FUNCTION_BLOCK FB_Beckhoff_EL5152
VAR_INPUT
	nValue1		: UINT;
	nValue2		: UINT;
END_VAR
VAR
	nControl1		AT %I* : UINT;
	nSetCounter1	AT %I* : UINT;
	nControl2		AT %I* : UINT;
	nSetCounter2	AT %I* : UINT;
	
	nStatus1		AT %Q* : UINT;
	nCounter1		AT %Q* : UINT;	
	nPeriod1    	AT %Q* : UDINT;
	nStatus2		AT %Q* : UINT;
	nCounter2		AT %Q* : UINT;
	nPeriod2    	AT %Q* : UDINT;
END_VAR

nStatus1.2 := nControl1.2;
nStatus2.2 := nControl2.2;

nCounter1 := nValue1;
nCounter2 := nValue2;

PROPERTY INTERNAL Control1 : UINT
SET
nControl1 := Control1;
END_SET
END_PROPERTY

PROPERTY INTERNAL Control2 : UINT
SET
nControl2 := Control2;
END_SET
END_PROPERTY

PROPERTY INTERNAL Counter1 : UINT
GET
Counter1 := nCounter1;
END_GET
END_PROPERTY

PROPERTY INTERNAL Counter2 : UINT
GET
Counter2 := nCounter2;
END_GET
END_PROPERTY

PROPERTY INTERNAL Period1 : UDINT
GET
Period1 := nPeriod1;
END_GET
END_PROPERTY

PROPERTY INTERNAL Period2 : UDINT
GET
Period2 := nPeriod2;
END_GET
END_PROPERTY

PROPERTY INTERNAL SetCounter1 : UINT
SET
nSetCounter1 := SetCounter1;
END_SET
END_PROPERTY

PROPERTY INTERNAL SetCounter2 : UINT
SET
nSetCounter2 := SetCounter2;
END_SET
END_PROPERTY

PROPERTY INTERNAL Status1 : UINT
GET
Status1 := nStatus1;
END_GET
END_PROPERTY

PROPERTY INTERNAL Status2 : UINT
GET
Status2 := nStatus2;
END_GET
END_PROPERTY

END_FUNCTION_BLOCK

(* stored: Version 1.1.0.1, ProductVersion 3.1.4024.12
   POU FB_Beckhoff_EL5152: Id {08baf088-2cf3-00bf-18c7-0387cec0c836}, SpecialFunc None
   Property Control1: Id {5c550402-bb0e-0ef9-0fec-73e14d2bbe4d}
   Set Set: Id {5ba60a83-acbe-0e98-31b5-a65c95cf5871}
   Property Control2: Id {f58e2f72-8d03-0b2d-15ce-8c78cfb46d19}
   Set Set: Id {5db5adfd-c3a6-0ac0-1eea-674a8bd0d24d}
   Property Counter1: Id {03127839-0093-03b2-0a6f-88166eb755f6}
   Get Get: Id {1ff40a2f-399d-0c65-15d8-0c3b4f2bcaeb}
   Property Counter2: Id {1854e639-ce6e-0901-076f-d57c64553137}
   Get Get: Id {3a7e0597-34bc-0eb5-0cc1-6255b4e03aaa}
   Property Period1: Id {1edf4574-7688-0a50-3510-8b9139b06165}
   Get Get: Id {bf0a7ae9-cbb6-0e81-047c-08773cbf0346}
   Property Period2: Id {09c7bfb3-9853-026e-3a6b-f81044b48193}
   Get Get: Id {56d16da8-379c-07e3-0b55-a85960b1f340}
   Property SetCounter1: Id {c25386e8-0be0-089c-3d08-5b0e80051126}
   Set Set: Id {b6324605-4dbc-0558-0ebc-4a9b3bcfda61}
   Property SetCounter2: Id {0e828313-bfa5-07ef-21f8-30993f027f98}
   Set Set: Id {a771431d-a0ee-034f-3d38-dbb5266e4a22}
   Property Status1: Id {aa2f335b-fbd1-0d43-01b9-27a2839cbdf2}
   Get Get: Id {967fca19-9e28-02b2-0a65-10b2dc3c998f}
   Property Status2: Id {82aa976b-c4e4-0291-378f-ade7c5039ac7}
   Get Get: Id {e014c008-b064-08f2-2379-4678fa2c02cc} *)
